PROGRAM MAIN
VAR
END_VAR

END_PROGRAM

(* stored: Version 1.1.0.1
   POU MAIN: Id {7a344413-1766-4f1a-948d-e4501bfe093c} *)
